// Mitsubishi GX Works2 project: Class5_IL&BIT&WORD(STEP)   PLC: Q03UD

PROGRAM MAIN
0     END
END_PROGRAM

PROGRAM ILSTEP
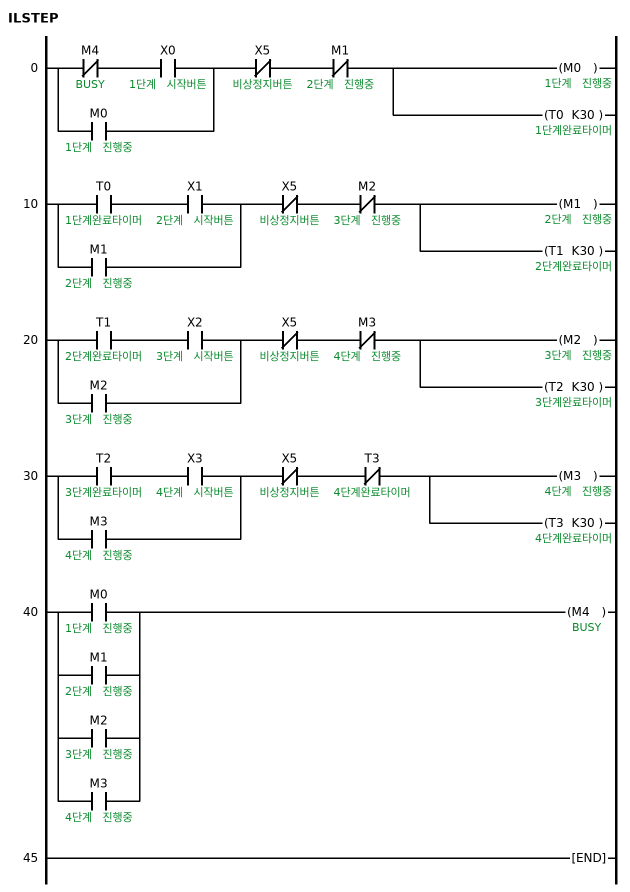
0     LDI     M4  ; BUSY
      AND     X0  ; 1단계   시작버튼
      OR      M0  ; 1단계   진행중
      ANI     X5  ; 비상정지버튼
      ANI     M1  ; 2단계   진행중
      OUT     M0  ; 1단계   진행중
      OUT     T0 K30  ; 1단계완료타이머
10    LD      T0  ; 1단계완료타이머
      AND     X1  ; 2단계   시작버튼
      OR      M1  ; 2단계   진행중
      ANI     X5  ; 비상정지버튼
      ANI     M2  ; 3단계   진행중
      OUT     M1  ; 2단계   진행중
      OUT     T1 K30  ; 2단계완료타이머
20    LD      T1  ; 2단계완료타이머
      AND     X2  ; 3단계   시작버튼
      OR      M2  ; 3단계   진행중
      ANI     X5  ; 비상정지버튼
      ANI     M3  ; 4단계   진행중
      OUT     M2  ; 3단계   진행중
      OUT     T2 K30  ; 3단계완료타이머
30    LD      T2  ; 3단계완료타이머
      AND     X3  ; 4단계   시작버튼
      OR      M3  ; 4단계   진행중
      ANI     X5  ; 비상정지버튼
      ANI     T3  ; 4단계완료타이머
      OUT     M3  ; 4단계   진행중
      OUT     T3 K30  ; 4단계완료타이머
40    LD      M0  ; 1단계   진행중
      OR      M1  ; 2단계   진행중
      OR      M2  ; 3단계   진행중
      OR      M3  ; 4단계   진행중
      OUT     M4  ; BUSY
45    END
END_PROGRAM

PROGRAM BITSTEP
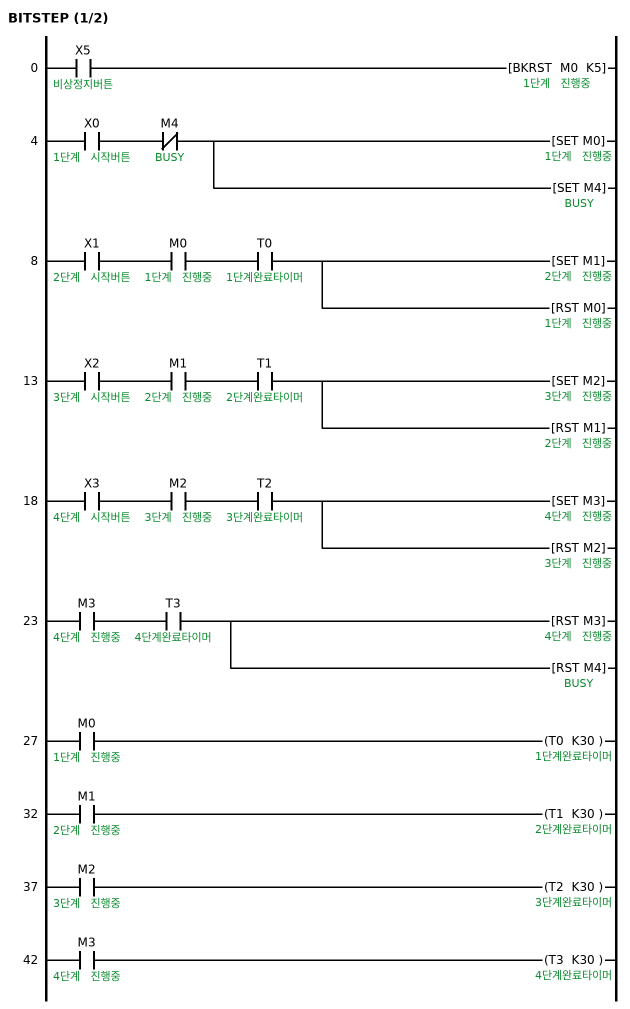
0     LD      X5  ; 비상정지버튼
      BKRST   M0 K5  ; 1단계   진행중
4     LD      X0  ; 1단계   시작버튼
      ANI     M4  ; BUSY
      SET     M0  ; 1단계   진행중
      SET     M4  ; BUSY
8     LD      X1  ; 2단계   시작버튼
      AND     M0  ; 1단계   진행중
      AND     T0  ; 1단계완료타이머
      SET     M1  ; 2단계   진행중
      RST     M0  ; 1단계   진행중
13    LD      X2  ; 3단계   시작버튼
      AND     M1  ; 2단계   진행중
      AND     T1  ; 2단계완료타이머
      SET     M2  ; 3단계   진행중
      RST     M1  ; 2단계   진행중
18    LD      X3  ; 4단계   시작버튼
      AND     M2  ; 3단계   진행중
      AND     T2  ; 3단계완료타이머
      SET     M3  ; 4단계   진행중
      RST     M2  ; 3단계   진행중
23    LD      M3  ; 4단계   진행중
      AND     T3  ; 4단계완료타이머
      RST     M3  ; 4단계   진행중
      RST     M4  ; BUSY
27    LD      M0  ; 1단계   진행중
      OUT     T0 K30  ; 1단계완료타이머
32    LD      M1  ; 2단계   진행중
      OUT     T1 K30  ; 2단계완료타이머
37    LD      M2  ; 3단계   진행중
      OUT     T2 K30  ; 3단계완료타이머
42    LD      M3  ; 4단계   진행중
      OUT     T3 K30  ; 4단계완료타이머
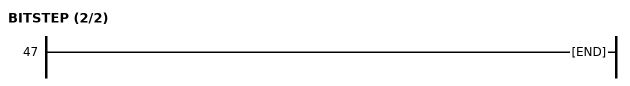
47    END
END_PROGRAM

PROGRAM WORDSTEP
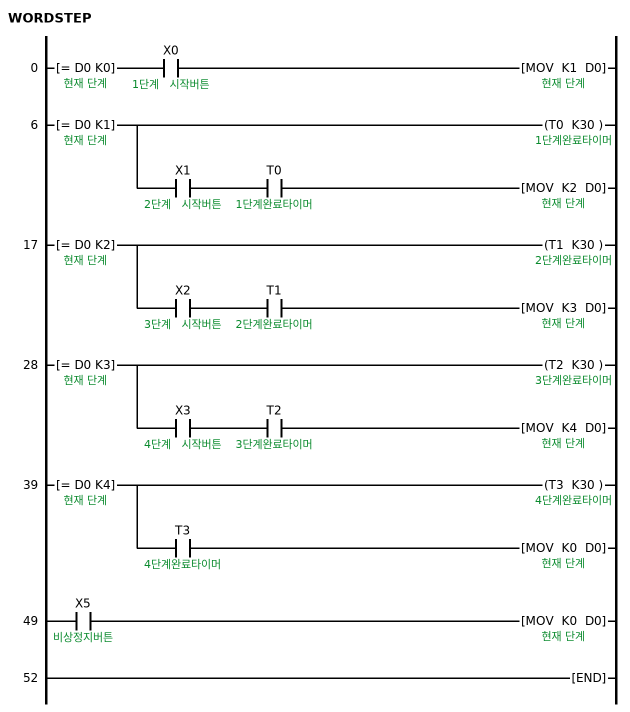
0     LD=     D0 K0  ; 현재 단계
      AND     X0  ; 1단계   시작버튼
      MOV     K1 D0
6     LD=     D0 K1  ; 현재 단계
      OUT     T0 K30  ; 1단계완료타이머
      AND     X1  ; 2단계   시작버튼
      AND     T0  ; 1단계완료타이머
      MOV     K2 D0
17    LD=     D0 K2  ; 현재 단계
      OUT     T1 K30  ; 2단계완료타이머
      AND     X2  ; 3단계   시작버튼
      AND     T1  ; 2단계완료타이머
      MOV     K3 D0
28    LD=     D0 K3  ; 현재 단계
      OUT     T2 K30  ; 3단계완료타이머
      AND     X3  ; 4단계   시작버튼
      AND     T2  ; 3단계완료타이머
      MOV     K4 D0
39    LD=     D0 K4  ; 현재 단계
      OUT     T3 K30  ; 4단계완료타이머
      AND     T3  ; 4단계완료타이머
      MOV     K0 D0
49    LD      X5  ; 비상정지버튼
      MOV     K0 D0
52    END
END_PROGRAM
